PROGRAM light
VAR
	light : BOOL;
	Lamp :BOOL;
END_VAR

light := Lamp;

END_PROGRAM

(* stored: Version 1.1.0.1, ProductVersion 3.1.4024.12
   POU light: Id {7e51ae7d-a41c-4121-9761-96be3489b038}, SpecialFunc None *)
